FUNCTION_BLOCK FB_ScopeServerSample
VAR_INPUT
	sNetId					: STRING	:='';	
    bExternalTriggerEvent	: BOOL 		:= FALSE; //Rising edge start recording, falling edge stop and save
	sConfigFile				: STRING(80); //.tcscopex
	sSaveFile				: STRING(80); //.svdx
END_VAR
VAR_OUTPUT
    bBusy					: BOOL 		:= FALSE;
    bError					: BOOL 		:= FALSE;
    nErrorId				: UDINT 	:= 0;	
END_VAR
VAR

    bDone					: BOOL 		:= FALSE;	

    fbScopeServerControl	: FB_ScopeServerControl;
    eReqState				: E_ScopeServerState := SCOPE_SERVER_IDLE;
	
    eState					: (IDLE,RECORDING,SAVING,DISCONNECTING,ERROR,RESETING);
END_VAR

CASE eState OF
	IDLE:
		bBusy	:=FALSE;
		IF bExternalTriggerEvent THEN
			bBusy			:= TRUE;
	    	eReqState 		:= SCOPE_SERVER_START;
	    	eState 			:= RECORDING;	
		END_IF
	
	RECORDING:	
		IF fbScopeServerControl.bDone THEN
	    	IF NOT bExternalTriggerEvent THEN
	    	    eReqState 		:= SCOPE_SERVER_SAVE;
	    	    eState 			:= SAVING;
	    	END_IF
		ELSIF fbScopeServerControl.bError THEN
			eState	:=ERROR;		
		END_IF
		
	SAVING:
	    IF fbScopeServerControl.bDone THEN
	        eReqState 		:= SCOPE_SERVER_DISCONNECT;
			eState			:= DISCONNECTING;
		ELSIF fbScopeServerControl.bError THEN
			eState	:=ERROR;		
		END_IF
		
	DISCONNECTING:
		IF fbScopeServerControl.bDone THEN
	       eState := IDLE;
		ELSIF fbScopeServerControl.bError THEN
			eState	:=ERROR;				   
	    END_IF		
		
	ERROR:
		bBusy			:= FALSE;
		IF NOT bExternalTriggerEvent THEN
			bBusy			:= TRUE;
			eReqState 		:= SCOPE_SERVER_RESET;
			eState			:= DISCONNECTING;
		END_IF
		
	RESETING:
		IF fbScopeServerControl.bDone OR fbScopeServerControl.bError THEN
	       	eReqState 		:= SCOPE_SERVER_IDLE;
			eState			:= IDLE; 
	    END_IF		
		
END_CASE


fbScopeServerControl( sNetId		:= '5.119.159.52.1.1',
                      eReqState		:= eReqState,
                      sConfigFile	:= sConfigFile,
                      sSaveFile		:= sSaveFile,
                      tTimeout		:= T#2S,
                      bBusy			=>,
                      bDone			=>bDone,
                      bError		=>bError,
                      nErrorId		=>nErrorId);

END_FUNCTION_BLOCK

(* stored: Version 1.1.0.1, ProductVersion 3.1.4024.12
   POU FB_ScopeServerSample: Id {e5cd026f-7b76-02ad-080f-a47ceddb5bba}, SpecialFunc None *)
